PROGRAM UpdateSync
VAR
	fbSqlDatabase : FB_SQLDatabaseEvt(sNetID := '', tTimeout := T#5S);
	fbSqlCommand : FB_SQLCommandEvt(sNetID := '', tTimeout := T#5S);
	myDBID: UDINT := 1;
	sTableName: STRING := 'Data';
	sCmd: STRING(1000);
	
	tcMessage1 : I_TcMessage;
	tcMessage2 : I_TcMessage;
	
	bFirstScan: BOOL := TRUE;
END_VAR

IF (bFirstScan) THEN
	IF fbSqlDatabase.Connect(myDBID) THEN
		bFirstScan := FALSE;
		IF fbSqlDatabase.bError THEN
			tcMessage1:= fbSqlDatabase.ipTcResult;
			bFirstScan := TRUE;
		END_IF
	END_IF
END_IF

IF GlobalData.bRemotePosted THEN
	CreateUpdate();
		
	IF fbSqlDatabase.CreateCmd(ADR(fbSqlCommand)) THEN
		IF fbSqlDatabase.bError THEN
			tcMessage1:= fbSqlDatabase.ipTcResult;
		END_IF
	END_IF
		
	IF fbSQLCommand.Execute(ADR(sCmd), LEN(sCmd)) THEN
		IF fbSQLCommand.bError THEN
			tcMessage2 := fbSQLCommand.ipTcResult;
		END_IF
		GlobalData.bRemotePosted := FALSE;
		GlobalData.blocalUpdated := TRUE;
		GlobalData.bMeasure := FALSE;
	END_IF
END_IF

ACTION CreateUpdate:
sCmd := 'UPDATE ';
sCmd := concat(sCmd, sTableName);
sCmd := concat(sCmd, ' SET Sync=');
sCmd := concat(sCmd, BOOL_TO_STRING(TRUE));
sCmd := concat(sCmd, ' WHERE Id=');
sCmd := concat(sCmd, LINT_TO_STRING(GlobalData.aReadStruct.iId));
END_ACTION

END_PROGRAM

(* stored: Version 1.1.0.1, ProductVersion 3.1.4024.4
   POU UpdateSync: Id {fbede189-66e5-4c6c-89b0-805380f05e5b}, SpecialFunc None
   Action CreateUpdate: Id {662f267f-a8f2-449b-a2ef-87a7054b0c20} *)
